{attribute 'qualified_only'}
{attribute 'strict'}
{attribute 'to_string'}
TYPE E_ScrewdriverErrorCode :
(
    None                       := 16#0000,
    ProcessFaultWithoutDetail  := 16#B600,
    PositionTimeout            := 16#B601,
    ScrewdriverCommandFailed   := 16#B602,
    AdjustmentCommandFailed    := 16#B603
) UDINT;
END_TYPE

(* stored: Version 1.1.0.1, ProductVersion 3.1.4026.20
   DUT E_ScrewdriverErrorCode: Id {fa78781e-3388-47b8-b16e-d3250440916a} *)
